PROGRAM TEST_AXIS
VAR
	fbRunAxis : POINTER TO RunAxis := ADR(GVL.axisControls[1]);
	
	ptCommand1 : POINTER TO CommandBlockGeneric := ADR(GVL.commandBlocks[1]);
	ptCommand2 : POINTER TO CommandBlockGeneric := ADR(GVL.commandBlocks[2]);
	
	state : INT;
	bDone : BOOL;
END_VAR

fbRunAxis^(); //service running


//pattern 1
CASE state OF
	0:
	fbRunAxis^.ExecuteCommandBlock(ptBlock:=ptCommand1,
		execute:= NOT bDone,
		bufferIndex:=1,
		done=> bDone);
	IF bDone THEN
		bDone := FALSE;
		state :=1;
	END_IF
	1:
	fbRunAxis^.ExecuteCommandBlock(ptBlock:=ptCommand2,
		execute:= NOT bDone,
		bufferIndex:=1,
		done=> bDone);
	IF bDone THEN
		bDone := FALSE;
		state :=0;
	END_IF
END_CASE

END_PROGRAM

(* stored: Version 1.1.0.1, ProductVersion 3.1.4020.12
   POU TEST_AXIS: Id {98ddbbdb-ba71-4026-957c-5163f7a8a335}, SpecialFunc None *)
